{attribute 'GeneratedUsingTerminal: EL3182-0000-0016'}
{attribute addProperty BoxType "EL3182-0000-0016"}
{attribute addProperty Id "EtcSlaveTerminalBaseCh_1Ch_1_A1FAE75910Ch_2Ch_2_D9CD36D210WcStateAT %I*WcState_9091E0EB2InfoDataAT %I*InfoData_90184F0C16"}
{attribute addProperty CRC "3372437287"}
{attribute addProperty Size "38"}
TYPE EL3182_C9034F27 EXTENDS EtcSlaveTerminalBase :
STRUCT
	{attribute addProperty Name "Ch_1"}
	Ch_1 : Ch_1_A1FAE759;
	{attribute addProperty Name "Ch_2"}
	Ch_2 : Ch_2_D9CD36D2;
	{attribute addProperty Name "WcState"}
	WcState : WcState_9091E0EB;
	{attribute addProperty Name "InfoData"}
	InfoData : InfoData_90184F0C;
END_STRUCT
END_TYPE

(* stored: Version 1.2.0.0, ProductVersion 3.1.4024.9
   DUT EL3182_C9034F27: Id {69f399e0-191f-46bc-87df-5b4125e09ac7} *)
